FUNCTION_BLOCK FB_RealControlBox IMPLEMENTS I_ControlBox
VAR_INPUT
END_VAR
VAR_OUTPUT
END_VAR
VAR
END_VAR

METHOD Joystick
VAR_INPUT
	eMode 	: E_Mode;
	eStatus : E_Status;
END_VAR
VAR_OUTPUT
	fJoystickY : LREAL;
END_VAR
IF eMode = E_Mode.Manual AND eStatus = E_Status.Running THEN
	fJoystickY := G_Sensors.fJoystickY;
ELSE
	fJoystickY := 0.0;
END_IF
END_METHOD

METHOD Lamps 
VAR_INPUT
	eMode 	: E_Mode;
	eStatus : E_Status;
END_VAR
IF eStatus = E_Status.Running AND NOT(eMode = E_Mode.Off) THEN
	G_Outputs.bGreenLight :=  TRUE;
ELSE
	G_Outputs.bGreenLight :=  FALSE;
END_IF

IF eStatus = E_Status.Fault  AND NOT(eMode = E_Mode.Off) THEN
	G_Outputs.bRedLight :=  TRUE;
ELSE
	G_Outputs.bRedLight :=  FALSE;
END_IF
END_METHOD

METHOD ModeSelector 
VAR_INPUT
END_VAR
VAR_OUTPUT
	eMode : E_Mode;
END_VAR
CASE eMode OF 
	E_Mode.Off:	
		IF G_Inputs.bManualModeSelector AND NOT(G_Inputs.bAutoModeSelector) THEN	
			eMode := E_Mode.Manual;
		END_IF
		
		IF G_Inputs.bAutoModeSelector AND NOT(G_Inputs.bManualModeSelector) THEN	
			eMode := E_Mode.Auto;
		END_IF

	E_Mode.Manual: 
		IF NOT(G_Inputs.bManualModeSelector) AND NOT(G_Inputs.bManualModeSelector) THEN	
			eMode := E_Mode.Off;
		END_IF
		
		IF G_Inputs.bAutoModeSelector AND NOT(G_Inputs.bManualModeSelector) THEN	
			eMode := E_Mode.Auto;
		END_IF
	
	E_Mode.Auto:
		IF NOT(G_Inputs.bManualModeSelector) AND NOT(G_Inputs.bManualModeSelector) THEN	
			eMode := E_Mode.Off;
		END_IF
		
		IF G_Inputs.bManualModeSelector AND NOT(G_Inputs.bAutoModeSelector) THEN	
			eMode := E_Mode.Manual;
		END_IF	
ELSE 	
	eMode := E_Mode.Off;
END_CASE
END_METHOD

METHOD PushButtons
VAR_INPUT
	eMode 	: E_Mode;
	eStatus : E_Status;
END_VAR
VAR_OUTPUT
	bStart : BOOL;
	bStop : BOOL;
END_VAR
IF NOT(eMode = E_Mode.Off) AND (NOT(eStatus = E_Status.Fault) OR (eStatus = E_Status.Off)) THEN 
	bStart := G_Inputs.bStartButton;
	bStop := G_Inputs.bStopButton;
ELSE
	bStart := FALSE;
	bStop := FALSE;
END_IF
END_METHOD

END_FUNCTION_BLOCK

(* stored: Version 1.1.0.1, ProductVersion 3.1.4024.10
   POU FB_RealControlBox: Id {37de488e-61db-47f0-ae9a-a602c45471dd}, SpecialFunc None
   Method Joystick: Id {969d1bf9-8f4a-4ed0-b706-e8d8185bf738}
   Method Lamps: Id {4fdeda89-2fc2-4bda-9219-00e0aed099ce}
   Method ModeSelector: Id {c1118847-ecf0-4ef4-a589-62e6a17557ee}
   Method PushButtons: Id {d7dda8b1-708c-4ae4-b6f1-5856535cda99} *)
